FUNCTION_BLOCK EL3024
VAR
	_io : EL3xx4_Data;
	{attribute addProperty Name "WcState"}
	_wcState : WcStateInputToggle;
	{attribute addProperty Name "Info data"}
	_infoData : InfoDataAds;
END_VAR

PROPERTY IO : REFERENCE TO EL3xx4_Data
GET
IO REF= _io;
END_GET
END_PROPERTY

PROPERTY WcState : REFERENCE TO WcStateInputToggle
GET
WcState REF= _wcState;
END_GET
END_PROPERTY

END_FUNCTION_BLOCK

(* stored: Version 1.1.0.1, ProductVersion 3.1.4024.9
   POU EL3024: Id {cbccfe41-aa0d-0f8b-371a-571f380a127f}, SpecialFunc None
   Property IO: Id {0cba8dcf-b089-032d-0de4-50909b757fc5}
   Get Get: Id {dc0bcd90-5533-0a9b-3352-243834d44289}
   Property WcState: Id {265d2cd1-6dc2-060e-15ec-8fc26cdfd247}
   Get Get: Id {eb994134-112b-065a-178a-3128de462aa1} *)
